Fanuc KAREL source: kt00306.KL

-- PROVISIONAL review KL for V770-1; original PC SHA256 ddcc08b1164fe1b7537d7b020509c81c626cd260070e99268befdd9c920caafe
-- Incomplete behavior may be omitted. Consult companion uncertainty JSON. Do not deploy.
PROGRAM KT00306
%NOLOCKGROUP
VAR
  OUT : BOOLEAN
-- UNRESOLVED_DECL Y1 type=002018
-- UNRESOLVED_DECL H2 type=002017
BEGIN
  -- UNRESOLVED_PC offsets 5-19; opcodes 2E,22,9D,33,B2
  -- UNRESOLVED_PC offsets 24-38; opcodes 2E,22,9D,33,B4
  -- UNRESOLVED_PC offsets 43-68; opcodes 22,9D,33,B1,22,9D,33,B3,58,23
  -- UNRESOLVED_PC offsets 73-77; opcodes 7F
END KT00306
